# EPICS substitutions: iocs/iocTest/boxTestApp/Db/boxTestApp.substitutions
file master.db
{
    pattern {P, S, VADDR, PORT}
    {"ECTEST", "", "999", "ECAT0"}

}
file el3702.db
{
}
